{attribute 'GeneratedUsingTerminal: KL9900-0055'}
{attribute addProperty BoxType "KL9900-0055"}
{attribute addProperty Id "Channel_1AT %Q*Channel_7DE261950"}
{attribute addProperty CRC "3918635876"}
{attribute addProperty Size "0"}
TYPE KL_E991A364 :
STRUCT
	{attribute addProperty Name "Channel_1"}
	Channel_1 : Channel_7DE26195;
END_STRUCT
END_TYPE

(* stored: Version 1.2.0.0, ProductVersion 3.1.4024.9
   DUT KL_E991A364: Id {2990ba60-ef88-4232-a939-eb9cf5f57706} *)
